// TwinCAT 3 PLC project MR1K4_PLC
// ProgramVersion: 3.1.4022.7
// libraries:
//   Tc2_SerialCom, * (Beckhoff Automation GmbH)
//   Tc2_Standard, * (Beckhoff Automation GmbH)
//   Tc2_System, * (Beckhoff Automation GmbH)
//   Tc2_Utilities, * (Beckhoff Automation GmbH)
//   Tc3_Module, * (Beckhoff Automation GmbH)
//   lcls-twincat-motion,1.1.0,SLAC
//   lcls-twincat-optics,0.0.0,SLAC
// project tree:
//   GVLs/ GVL_COM_Buffers.TcGVL (not stored), GVL_M1K4.TcGVL, GVL_M1K4_Constants.TcGVL (not stored), GVL_SerialIO.TcGVL
//   / PiezoDriver.TcTTO, PlcTask.TcTTO, SerialIO.TcTTO
//   POUs/ Main.TcPOU
//   POUs/Serial Comm/ PiezoSerial.TcPOU, P_Serial_Com.TcPOU
// real-time tasks:
//   TASK PlcTask: cycle T#10ms, priority 20, ADS port 350
//   TASK PiezoDriver: cycle T#1ms, priority 3, ADS port 351
//   TASK SerialIO: cycle T#2ms, priority 1, ADS port 352
// motion (NC):
//   TASK NC-Task 1 SAF: cycle T#2ms, priority 4, ADS port 501
//   TASK NC-Task 1 SVB: cycle T#10ms, priority 8, ADS port 511
//   AXIS M1K4-Yup (id 1)
//     General: UnitName=um
//     Dynamic: Acceleration=200, Deceleration=200, DelayTime=0.008
//     Velo: Maximum=200
//     OtherSettings: AllowMotionCmdToSlave=true
//     encoder EncType=29
//       EncPara: ScaleFactorNumerator=0.001, MaxCount=#xffffffff
//         SoftEndMinControl: Enable=true, Range=2700
//         SoftEndMaxControl: Enable=true, Range=27000
//         Inc: RefSoftSyncMask=#x0000ffff
//     drive DrvType=24
//       DrvPara: Inverse=true
//         Analog: VeloReferenz=488.28125, ScaleFactorActTorque=0.1
//         TimeComp: TaskDelayCycles=1
//     controller CtrType=2
//       CtrPara: PriorControlFactor=1
//         PosDiffControl: Range=100
//         PID: PosKp=50, PosExtKp=10, DeadBandPosition=0.3
//         Observer: BandWidth=20
//   AXIS M1K4-Ydwn (id 2)
//     General: UnitName=um
//     Dynamic: Acceleration=200, Deceleration=200, DelayTime=0.008
//     Velo: Maximum=200
//     OtherSettings: AllowMotionCmdToSlave=true
//     encoder EncType=29
//       EncPara: ScaleFactorNumerator=0.001, MaxCount=#xffffffff
//         SoftEndMinControl: Enable=true, Range=2400
//         SoftEndMaxControl: Enable=true, Range=26700
//         Inc: RefSoftSyncMask=#x0000ffff
//     drive DrvType=24
//       DrvPara: Inverse=true
//         Analog: VeloReferenz=488.28125, ScaleFactorActTorque=0.1
//         TimeComp: TaskDelayCycles=1
//     controller CtrType=2
//       CtrPara: PriorControlFactor=1
//         PosDiffControl: Range=100
//         PID: PosKp=50, PosExtKp=10, DeadBandPosition=0.3
//         Observer: BandWidth=20
//   AXIS M1K4-Xup (id 3)
//     General: UnitName=um
//     Dynamic: Acceleration=2000, Deceleration=2000, DelayTime=0.008
//     Velo: Maximum=1000
//     OtherSettings: AllowMotionCmdToSlave=true
//     encoder EncType=29
//       EncPara: ScaleFactorNumerator=0.001, MaxCount=#xffffffff
//         SoftEndMinControl: Enable=true, Range=23400
//         SoftEndMaxControl: Enable=true, Range=25700
//         Inc: RefSoftSyncMask=#x0000ffff
//     drive DrvType=24
//       Analog: VeloReferenz=1220.703125, ScaleFactorActTorque=0.1
//       TimeComp: TaskDelayCycles=1
//     controller CtrType=2
//       CtrPara: PriorControlFactor=1
//         PosDiffControl: Range=100
//         PID: PosKp=50, PosExtKp=50, DeadBandPosition=0.4
//         Observer: BandWidth=20
//   AXIS M1K4-Xdwn (id 4)
//     General: UnitName=um
//     Dynamic: Acceleration=2000, Deceleration=2000, DelayTime=0.008
//     Velo: Maximum=1000
//     OtherSettings: AllowMotionCmdToSlave=true
//     encoder EncType=29
//       EncPara: ScaleFactorNumerator=0.001, MaxCount=#xffffffff
//         SoftEndMinControl: Enable=true, Range=23400
//         SoftEndMaxControl: Enable=true, Range=25800
//         Inc: RefSoftSyncMask=#x0000ffff
//     drive DrvType=24
//       DrvPara: Inverse=true
//         Analog: VeloReferenz=1220.703125, ScaleFactorActTorque=0.1
//         TimeComp: TaskDelayCycles=1
//     controller CtrType=2
//       CtrPara: PriorControlFactor=1
//         PosDiffControl: Range=100
//         PID: PosKp=50, PosExtKp=50, DeadBandPosition=0.4
//         Observer: BandWidth=20
//   AXIS M1K4-Pitch (id 5)
//     General: UnitName=urad
//     Dynamic: Acceleration=390, Deceleration=390, DelayTime=0.008
//     Velo: Maximum=150
//     OtherSettings: AllowMotionCmdToSlave=true
//     encoder EncType=29
//       EncPara: ScaleFactorNumerator=0.001949317739, MaxCount=#xffffffff
//         SoftEndMinControl: Enable=true, Range=17200
//         SoftEndMaxControl: Enable=true, Range=21800
//         Inc: RefSoftSyncMask=#x0000ffff
//     drive DrvType=24
//       Analog: VeloReferenz=761.4522417, ScaleFactorActTorque=0.1
//       TimeComp: TaskDelayCycles=1
//     controller CtrType=2
//       CtrPara: PriorControlFactor=1
//         PosDiffControl: Range=150
//         PID: PosExtKp=1, DeadBandPosition=0.25
//         Observer: BandWidth=20
//   AXIS M1K4-Bender (id 6)
//     General: UnitName=um
//     Dynamic: Acceleration=100, Deceleration=100, DelayTime=0.008
//     Velo: Maximum=190
//     OtherSettings: AllowMotionCmdToSlave=true
//     encoder EncType=29
//       EncPara: ScaleFactorNumerator=0.001, MaxCount=#xffffffff
//         Inc: RefSoftSyncMask=#x0000ffff
//     drive DrvType=24
//       Analog: VeloReferenz=195.3125, ScaleFactorActTorque=0.1
//       TimeComp: TaskDelayCycles=1
//     controller CtrType=2
//       CtrPara: PriorControlFactor=1
//         PID: PosKp=10, PosExtKp=1, DeadBandPosition=0.04
//         Observer: BandWidth=20
// I/O:
//   DEVICE Device 1 (EtherCAT), AmsNetId 172.21.92.63.2.1
//     Term 1 (EK1200)
// variable links:
//   (this object) <-> Device 1 (EtherCAT)/Term 1 (EK1200)/Term 5 (EK1122)/Term 6 (EK1100)/EL5042_M1K4_Yupdwn
//     Enc/Inputs/In/nComState @bit 1 <-> WcState/InputToggle
//     Enc/Inputs/In/nComState <-> WcState/WcState
//     Enc/Inputs/In/nDataIn1 <-> FB Inputs Channel 1/Position
//     Enc/Inputs/In/nDataIn1 <-> FB Inputs Channel 2/Position
//     Enc/Inputs/In/nState1 @bit 12 <-> FB Inputs Channel 1/Status/Diag
//     Enc/Inputs/In/nState1 @bit 12 <-> FB Inputs Channel 2/Status/Diag
//     Enc/Inputs/In/nState1 @bit 1 <-> FB Inputs Channel 1/Status/Error
//     Enc/Inputs/In/nState1 @bit 1 <-> FB Inputs Channel 2/Status/Error
//     Enc/Inputs/In/nState1 @bit 14 <-> FB Inputs Channel 1/Status/Input cycle counter
//     Enc/Inputs/In/nState1 @bit 14 <-> FB Inputs Channel 2/Status/Input cycle counter
//     Enc/Inputs/In/nState1 @bit 2 <-> FB Inputs Channel 1/Status/Ready
//     Enc/Inputs/In/nState1 @bit 2 <-> FB Inputs Channel 2/Status/Ready
//     Enc/Inputs/In/nState1 @bit 13 <-> FB Inputs Channel 1/Status/TxPDO State
//     Enc/Inputs/In/nState1 @bit 13 <-> FB Inputs Channel 2/Status/TxPDO State
//     Enc/Inputs/In/nState1 <-> FB Inputs Channel 1/Status/Warning
//     Enc/Inputs/In/nState1 <-> FB Inputs Channel 2/Status/Warning
//   (this object) <-> Device 1 (EtherCAT)/Term 1 (EK1200)/Term 5 (EK1122)/Term 6 (EK1100)/EL7041-1000_M1K4_Yup
//     Drive/Inputs/In/nState1 @bit 3 <-> STM Status/Status/Error
//     Drive/Inputs/In/nState1 @bit 5 <-> STM Status/Status/Moving negative
//     Drive/Inputs/In/nState1 @bit 4 <-> STM Status/Status/Moving positive
//     Drive/Inputs/In/nState1 @bit 1 <-> STM Status/Status/Ready
//     Drive/Inputs/In/nState1 <-> STM Status/Status/Ready to enable
//     Drive/Inputs/In/nState1 @bit 6 <-> STM Status/Status/Torque reduced
//     Drive/Inputs/In/nState1 @bit 2 <-> STM Status/Status/Warning
//     Drive/Inputs/In/nState2 @bit 3 <-> STM Status/Status/Digital input 1
//     Drive/Inputs/In/nState2 @bit 4 <-> STM Status/Status/Digital input 2
//     Drive/Inputs/In/nState2 @bit 5 <-> STM Status/Status/Sync error
//     Drive/Inputs/In/nState2 @bit 7 <-> STM Status/Status/TxPDO Toggle
//     Drive/Inputs/In/nState4 @bit 1 <-> WcState/InputToggle
//     Drive/Inputs/In/nState4 <-> WcState/WcState
//     Drive/Outputs/Out/nCtrl1 <-> STM Control/Control/Enable
//     Drive/Outputs/Out/nCtrl1 @bit 2 <-> STM Control/Control/Reduce torque
//     Drive/Outputs/Out/nCtrl1 @bit 1 <-> STM Control/Control/Reset
//     Drive/Outputs/Out/nDataOut2[0] <-> STM Velocity/Velocity
//   (this object) <-> Device 1 (EtherCAT)/Term 1 (EK1200)/Term 5 (EK1122)/Term 6 (EK1100)/EL7041-1000_M1K4_Ydwn
//     Drive/Inputs/In/nState1 @bit 3 <-> STM Status/Status/Error
//     Drive/Inputs/In/nState1 @bit 5 <-> STM Status/Status/Moving negative
//     Drive/Inputs/In/nState1 @bit 4 <-> STM Status/Status/Moving positive
//     Drive/Inputs/In/nState1 @bit 1 <-> STM Status/Status/Ready
//     Drive/Inputs/In/nState1 <-> STM Status/Status/Ready to enable
//     Drive/Inputs/In/nState1 @bit 6 <-> STM Status/Status/Torque reduced
//     Drive/Inputs/In/nState1 @bit 2 <-> STM Status/Status/Warning
//     Drive/Inputs/In/nState2 @bit 3 <-> STM Status/Status/Digital input 1
//     Drive/Inputs/In/nState2 @bit 4 <-> STM Status/Status/Digital input 2
//     Drive/Inputs/In/nState2 @bit 5 <-> STM Status/Status/Sync error
//     Drive/Inputs/In/nState2 @bit 7 <-> STM Status/Status/TxPDO Toggle
//     Drive/Inputs/In/nState4 @bit 1 <-> WcState/InputToggle
//     Drive/Inputs/In/nState4 <-> WcState/WcState
//     Drive/Outputs/Out/nCtrl1 <-> STM Control/Control/Enable
//     Drive/Outputs/Out/nCtrl1 @bit 2 <-> STM Control/Control/Reduce torque
//     Drive/Outputs/Out/nCtrl1 @bit 1 <-> STM Control/Control/Reset
//     Drive/Outputs/Out/nDataOut2[0] <-> STM Velocity/Velocity
//   (this object) <-> Device 1 (EtherCAT)/Term 1 (EK1200)/Term 5 (EK1122)/Term 6 (EK1100)/EL5042_M1K4_Xupdwn
//     Enc/Inputs/In/nComState @bit 1 <-> WcState/InputToggle
//     Enc/Inputs/In/nComState <-> WcState/WcState
//     Enc/Inputs/In/nDataIn1 <-> FB Inputs Channel 1/Position
//     Enc/Inputs/In/nDataIn1 <-> FB Inputs Channel 2/Position
//     Enc/Inputs/In/nState1 @bit 12 <-> FB Inputs Channel 1/Status/Diag
//     Enc/Inputs/In/nState1 @bit 12 <-> FB Inputs Channel 2/Status/Diag
//     Enc/Inputs/In/nState1 @bit 1 <-> FB Inputs Channel 1/Status/Error
//     Enc/Inputs/In/nState1 @bit 1 <-> FB Inputs Channel 2/Status/Error
//     Enc/Inputs/In/nState1 @bit 14 <-> FB Inputs Channel 1/Status/Input cycle counter
//     Enc/Inputs/In/nState1 @bit 14 <-> FB Inputs Channel 2/Status/Input cycle counter
//     Enc/Inputs/In/nState1 @bit 2 <-> FB Inputs Channel 1/Status/Ready
//     Enc/Inputs/In/nState1 @bit 2 <-> FB Inputs Channel 2/Status/Ready
//     Enc/Inputs/In/nState1 @bit 13 <-> FB Inputs Channel 1/Status/TxPDO State
//     Enc/Inputs/In/nState1 @bit 13 <-> FB Inputs Channel 2/Status/TxPDO State
//     Enc/Inputs/In/nState1 <-> FB Inputs Channel 1/Status/Warning
//     Enc/Inputs/In/nState1 <-> FB Inputs Channel 2/Status/Warning
//   (this object) <-> Device 1 (EtherCAT)/Term 1 (EK1200)/Term 5 (EK1122)/Term 6 (EK1100)/EL7041-1000_M1K4_Xup
//     Drive/Inputs/In/nState1 @bit 3 <-> STM Status/Status/Error
//     Drive/Inputs/In/nState1 @bit 5 <-> STM Status/Status/Moving negative
//     Drive/Inputs/In/nState1 @bit 4 <-> STM Status/Status/Moving positive
//     Drive/Inputs/In/nState1 @bit 1 <-> STM Status/Status/Ready
//     Drive/Inputs/In/nState1 <-> STM Status/Status/Ready to enable
//     Drive/Inputs/In/nState1 @bit 6 <-> STM Status/Status/Torque reduced
//     Drive/Inputs/In/nState1 @bit 2 <-> STM Status/Status/Warning
//     Drive/Inputs/In/nState2 @bit 3 <-> STM Status/Status/Digital input 1
//     Drive/Inputs/In/nState2 @bit 4 <-> STM Status/Status/Digital input 2
//     Drive/Inputs/In/nState2 @bit 5 <-> STM Status/Status/Sync error
//     Drive/Inputs/In/nState2 @bit 7 <-> STM Status/Status/TxPDO Toggle
//     Drive/Inputs/In/nState4 @bit 1 <-> WcState/InputToggle
//     Drive/Inputs/In/nState4 <-> WcState/WcState
//     Drive/Outputs/Out/nCtrl1 <-> STM Control/Control/Enable
//     Drive/Outputs/Out/nCtrl1 @bit 2 <-> STM Control/Control/Reduce torque
//     Drive/Outputs/Out/nCtrl1 @bit 1 <-> STM Control/Control/Reset
//     Drive/Outputs/Out/nDataOut2[0] <-> STM Velocity/Velocity
//   (this object) <-> Device 1 (EtherCAT)/Term 1 (EK1200)/Term 5 (EK1122)/Term 6 (EK1100)/EL7041-1000_M1K4_Xdwn
//     Drive/Inputs/In/nState1 @bit 3 <-> STM Status/Status/Error
//     Drive/Inputs/In/nState1 @bit 5 <-> STM Status/Status/Moving negative
//     Drive/Inputs/In/nState1 @bit 4 <-> STM Status/Status/Moving positive
//     Drive/Inputs/In/nState1 @bit 1 <-> STM Status/Status/Ready
//     Drive/Inputs/In/nState1 <-> STM Status/Status/Ready to enable
//     Drive/Inputs/In/nState1 @bit 6 <-> STM Status/Status/Torque reduced
//     Drive/Inputs/In/nState1 @bit 2 <-> STM Status/Status/Warning
//     Drive/Inputs/In/nState2 @bit 3 <-> STM Status/Status/Digital input 1
//     Drive/Inputs/In/nState2 @bit 4 <-> STM Status/Status/Digital input 2
//     Drive/Inputs/In/nState2 @bit 5 <-> STM Status/Status/Sync error
//     Drive/Inputs/In/nState2 @bit 7 <-> STM Status/Status/TxPDO Toggle
//     Drive/Inputs/In/nState4 @bit 1 <-> WcState/InputToggle
//     Drive/Inputs/In/nState4 <-> WcState/WcState
//     Drive/Outputs/Out/nCtrl1 <-> STM Control/Control/Enable
//     Drive/Outputs/Out/nCtrl1 @bit 2 <-> STM Control/Control/Reduce torque
//     Drive/Outputs/Out/nCtrl1 @bit 1 <-> STM Control/Control/Reset
//     Drive/Outputs/Out/nDataOut2[0] <-> STM Velocity/Velocity
//   (this object) <-> Device 1 (EtherCAT)/Term 1 (EK1200)/Term 5 (EK1122)/Term 6 (EK1100)/EL5042_M1K4_PitchBender
//     Enc/Inputs/In/nComState @bit 1 <-> WcState/InputToggle
//     Enc/Inputs/In/nComState <-> WcState/WcState
//     Enc/Inputs/In/nDataIn1 <-> FB Inputs Channel 1/Position
//     Enc/Inputs/In/nDataIn1 <-> FB Inputs Channel 2/Position
//     Enc/Inputs/In/nState1 @bit 12 <-> FB Inputs Channel 1/Status/Diag
//     Enc/Inputs/In/nState1 @bit 12 <-> FB Inputs Channel 2/Status/Diag
//     Enc/Inputs/In/nState1 @bit 1 <-> FB Inputs Channel 1/Status/Error
//     Enc/Inputs/In/nState1 @bit 1 <-> FB Inputs Channel 2/Status/Error
//     Enc/Inputs/In/nState1 @bit 14 <-> FB Inputs Channel 1/Status/Input cycle counter
//     Enc/Inputs/In/nState1 @bit 14 <-> FB Inputs Channel 2/Status/Input cycle counter
//     Enc/Inputs/In/nState1 @bit 2 <-> FB Inputs Channel 1/Status/Ready
//     Enc/Inputs/In/nState1 @bit 2 <-> FB Inputs Channel 2/Status/Ready
//     Enc/Inputs/In/nState1 @bit 13 <-> FB Inputs Channel 1/Status/TxPDO State
//     Enc/Inputs/In/nState1 @bit 13 <-> FB Inputs Channel 2/Status/TxPDO State
//     Enc/Inputs/In/nState1 <-> FB Inputs Channel 1/Status/Warning
//     Enc/Inputs/In/nState1 <-> FB Inputs Channel 2/Status/Warning
//   (this object) <-> Device 1 (EtherCAT)/Term 1 (EK1200)/Term 5 (EK1122)/Term 6 (EK1100)/EL7041-1000_M1K4_PitchCoarse
//     Drive/Inputs/In/nState1 @bit 3 <-> STM Status/Status/Error
//     Drive/Inputs/In/nState1 @bit 5 <-> STM Status/Status/Moving negative
//     Drive/Inputs/In/nState1 @bit 4 <-> STM Status/Status/Moving positive
//     Drive/Inputs/In/nState1 @bit 1 <-> STM Status/Status/Ready
//     Drive/Inputs/In/nState1 <-> STM Status/Status/Ready to enable
//     Drive/Inputs/In/nState1 @bit 6 <-> STM Status/Status/Torque reduced
//     Drive/Inputs/In/nState1 @bit 2 <-> STM Status/Status/Warning
//     Drive/Inputs/In/nState2 @bit 3 <-> STM Status/Status/Digital input 1
//     Drive/Inputs/In/nState2 @bit 4 <-> STM Status/Status/Digital input 2
//     Drive/Inputs/In/nState2 @bit 5 <-> STM Status/Status/Sync error
//     Drive/Inputs/In/nState2 @bit 7 <-> STM Status/Status/TxPDO Toggle
//     Drive/Inputs/In/nState4 @bit 1 <-> WcState/InputToggle
//     Drive/Inputs/In/nState4 <-> WcState/WcState
//     Drive/Outputs/Out/nCtrl1 <-> STM Control/Control/Enable
//     Drive/Outputs/Out/nCtrl1 @bit 2 <-> STM Control/Control/Reduce torque
//     Drive/Outputs/Out/nCtrl1 @bit 1 <-> STM Control/Control/Reset
//     Drive/Outputs/Out/nDataOut2[0] <-> STM Velocity/Velocity
//   (this object) <-> Device 1 (EtherCAT)/Term 1 (EK1200)/Term 5 (EK1122)/Term 6 (EK1100)/EL7041-1000_M1K4_Bender
//     Drive/Inputs/In/nState1 @bit 3 <-> STM Status/Status/Error
//     Drive/Inputs/In/nState1 @bit 5 <-> STM Status/Status/Moving negative
//     Drive/Inputs/In/nState1 @bit 4 <-> STM Status/Status/Moving positive
//     Drive/Inputs/In/nState1 @bit 1 <-> STM Status/Status/Ready
//     Drive/Inputs/In/nState1 <-> STM Status/Status/Ready to enable
//     Drive/Inputs/In/nState1 @bit 6 <-> STM Status/Status/Torque reduced
//     Drive/Inputs/In/nState1 @bit 2 <-> STM Status/Status/Warning
//     Drive/Inputs/In/nState2 @bit 3 <-> STM Status/Status/Digital input 1
//     Drive/Inputs/In/nState2 @bit 4 <-> STM Status/Status/Digital input 2
//     Drive/Inputs/In/nState2 @bit 5 <-> STM Status/Status/Sync error
//     Drive/Inputs/In/nState2 @bit 7 <-> STM Status/Status/TxPDO Toggle
//     Drive/Inputs/In/nState4 @bit 1 <-> WcState/InputToggle
//     Drive/Inputs/In/nState4 <-> WcState/WcState
//     Drive/Outputs/Out/nCtrl1 <-> STM Control/Control/Enable
//     Drive/Outputs/Out/nCtrl1 @bit 2 <-> STM Control/Control/Reduce torque
//     Drive/Outputs/Out/nCtrl1 @bit 1 <-> STM Control/Control/Reset
//     Drive/Outputs/Out/nDataOut2[0] <-> STM Velocity/Velocity
//   MR1K4_PLC Instance <-> Device 1 (EtherCAT)/Term 1 (EK1200)/Term 5 (EK1122)/Term 6 (EK1100)/EL1004_M1K4_STO
//     PlcTask Inputs/Main.M1K4.fbRunHOMS.bSTOEnable1 <-> Channel 1/Input
//     PlcTask Inputs/Main.M1K4.fbRunHOMS.bSTOEnable2 <-> Channel 2/Input
//   MR1K4_PLC Instance <-> Device 1 (EtherCAT)/Term 1 (EK1200)/Term 5 (EK1122)/Term 6 (EK1100)/EL5042_M1K4_PitchBender
//     PlcTask Inputs/GVL_M1K4.M1K4_Pitch.diEncCnt <-> FB Inputs Channel 1/Position
//   MR1K4_PLC Instance <-> Device 1 (EtherCAT)/Term 1 (EK1200)/Term 5 (EK1122)/Term 6 (EK1100)/EL5042_M1K4_Xupdwn
//     PlcTask Inputs/Main.M1K4.fbRunHOMS.stXdwnEnc/Count <-> FB Inputs Channel 2/Position
//     PlcTask Inputs/Main.M1K4.fbRunHOMS.stXupEnc/Count <-> FB Inputs Channel 1/Position
//   MR1K4_PLC Instance <-> Device 1 (EtherCAT)/Term 1 (EK1200)/Term 5 (EK1122)/Term 6 (EK1100)/EL5042_M1K4_Yupdwn
//     PlcTask Inputs/Main.M1K4.fbRunHOMS.stYdwnEnc/Count <-> FB Inputs Channel 2/Position
//     PlcTask Inputs/Main.M1K4.fbRunHOMS.stYupEnc/Count <-> FB Inputs Channel 1/Position
//   MR1K4_PLC Instance <-> Device 1 (EtherCAT)/Term 1 (EK1200)/Term 5 (EK1122)/Term 6 (EK1100)/EL6001_M1K4_PitchFine
//     SerialIO Inputs/GVL_SerialIO.Serial_stComIn_M1K4/D[{0..21}] <-> COM Inputs/Data In {0..21}  (22 links)
//     SerialIO Inputs/GVL_SerialIO.Serial_stComIn_M1K4/Status <-> COM Inputs/Status
//     SerialIO Outputs/GVL_SerialIO.Serial_stComOut_M1K4/Ctrl <-> COM Outputs/Ctrl
//     SerialIO Outputs/GVL_SerialIO.Serial_stComOut_M1K4/D[{0..21}] <-> COM Outputs/Data Out {0..21}  (22 links)
//   MR1K4_PLC Instance <-> Device 1 (EtherCAT)/Term 1 (EK1200)/Term 5 (EK1122)/Term 6 (EK1100)/EL7041-1000_M1K4_Bender
//     PlcTask Inputs/Main.M6.bLimitBackwardEnable <-> STM Status/Status/Digital input 2
//     PlcTask Inputs/Main.M6.bLimitForwardEnable <-> STM Status/Status/Digital input 1
//   MR1K4_PLC Instance <-> Device 1 (EtherCAT)/Term 1 (EK1200)/Term 5 (EK1122)/Term 6 (EK1100)/EL7041-1000_M1K4_PitchCoarse
//     PlcTask Inputs/Main.M5.bLimitBackwardEnable <-> STM Status/Status/Digital input 2
//     PlcTask Inputs/Main.M5.bLimitForwardEnable <-> STM Status/Status/Digital input 1
//   MR1K4_PLC Instance <-> Device 1 (EtherCAT)/Term 1 (EK1200)/Term 5 (EK1122)/Term 6 (EK1100)/EL7041-1000_M1K4_Xdwn
//     PlcTask Inputs/Main.M4.bLimitBackwardEnable <-> STM Status/Status/Digital input 2
//     PlcTask Inputs/Main.M4.bLimitForwardEnable <-> STM Status/Status/Digital input 1
//   MR1K4_PLC Instance <-> Device 1 (EtherCAT)/Term 1 (EK1200)/Term 5 (EK1122)/Term 6 (EK1100)/EL7041-1000_M1K4_Xup
//     PlcTask Inputs/Main.M3.bLimitBackwardEnable <-> STM Status/Status/Digital input 2
//     PlcTask Inputs/Main.M3.bLimitForwardEnable <-> STM Status/Status/Digital input 1
//   MR1K4_PLC Instance <-> Device 1 (EtherCAT)/Term 1 (EK1200)/Term 5 (EK1122)/Term 6 (EK1100)/EL7041-1000_M1K4_Ydwn
//     PlcTask Inputs/Main.M2.bLimitBackwardEnable <-> STM Status/Status/Digital input 2
//     PlcTask Inputs/Main.M2.bLimitForwardEnable <-> STM Status/Status/Digital input 1
//   MR1K4_PLC Instance <-> Device 1 (EtherCAT)/Term 1 (EK1200)/Term 5 (EK1122)/Term 6 (EK1100)/EL7041-1000_M1K4_Yup
//     PlcTask Inputs/Main.M1.bLimitBackwardEnable <-> STM Status/Status/Digital input 2
//     PlcTask Inputs/Main.M1.bLimitForwardEnable <-> STM Status/Status/Digital input 1
//   MR1K4_PLC Instance <-> NC-Task 1 SAF/Axes/M1K4-Bender
//     PlcTask Inputs/Main.M6.Axis.NcToPlc <-> Outputs/ToPlc
//     PlcTask Outputs/Main.M6.Axis.PlcToNc <-> Inputs/FromPlc
//   MR1K4_PLC Instance <-> NC-Task 1 SAF/Axes/M1K4-Pitch
//     PlcTask Inputs/Main.M5.Axis.NcToPlc <-> Outputs/ToPlc
//     PlcTask Outputs/Main.M5.Axis.PlcToNc <-> Inputs/FromPlc
//   MR1K4_PLC Instance <-> NC-Task 1 SAF/Axes/M1K4-Xdwn
//     PlcTask Inputs/Main.M4.Axis.NcToPlc <-> Outputs/ToPlc
//     PlcTask Outputs/Main.M4.Axis.PlcToNc <-> Inputs/FromPlc
//   MR1K4_PLC Instance <-> NC-Task 1 SAF/Axes/M1K4-Xup
//     PlcTask Inputs/Main.M3.Axis.NcToPlc <-> Outputs/ToPlc
//     PlcTask Outputs/Main.M3.Axis.PlcToNc <-> Inputs/FromPlc
//   MR1K4_PLC Instance <-> NC-Task 1 SAF/Axes/M1K4-Ydwn
//     PlcTask Inputs/Main.M2.Axis.NcToPlc <-> Outputs/ToPlc
//     PlcTask Outputs/Main.M2.Axis.PlcToNc <-> Inputs/FromPlc
//   MR1K4_PLC Instance <-> NC-Task 1 SAF/Axes/M1K4-Yup
//     PlcTask Inputs/Main.M1.Axis.NcToPlc <-> Outputs/ToPlc
//     PlcTask Outputs/Main.M1.Axis.PlcToNc <-> Inputs/FromPlc

CONFIGURATION MR1K4_PLC
    RESOURCE PLC ON TwinCAT3
        TASK PiezoDriver(INTERVAL := T#1ms, PRIORITY := 3);
        TASK PlcTask(INTERVAL := T#10ms, PRIORITY := 20);
        TASK SerialIO(INTERVAL := T#2ms, PRIORITY := 1);
        PROGRAM PiezoSerial WITH PiezoDriver : PiezoSerial;
        PROGRAM MAIN WITH PlcTask : MAIN;
        PROGRAM P_Serial_Com WITH SerialIO : P_Serial_Com;
    END_RESOURCE
END_CONFIGURATION

// ---- GVLs/GVL_M1K4.TcGVL
{attribute 'qualified_only'}
VAR_GLOBAL
	// Pitch Mechanism:
	{attribute 'TcLinkTo' := '.diEncCnt:=TIIB[EL5042_M1K4_PitchBender]^FB Inputs Channel 1^Position'}
	M1K4_Pitch : HOMS_PitchMechanism := (ReqPosLimHi := 21700,
		                                 ReqPosLimLo := 17400,
		                                 diEncPosLimHi := 11132100,
		                                 diEncPosLimLo := 8926200);
END_VAR

// ---- GVLs/GVL_SerialIO.TcGVL
VAR_GLOBAL
	//Better have your inputs and outputs!
	// M1K4
	Serial_stComIn_M1K4   AT %I*	:	EL6inData22B (*KL6inData22B*);
	Serial_stComOut_M1K4  AT %Q*	:	EL6outData22B (*KL6outData22B*);
END_VAR

// ---- POUs/Serial Comm/PiezoSerial.TcPOU
PROGRAM PiezoSerial
VAR
	//PI Serial
	fbE621SerialDriver_M1K4 : FB_PI_E621_SerialDriver;
	rtInitParams_M1K4	:	R_TRIG;
	tonTimeoutRst_M1K4	: TON := (PT:=T#2S); //For timeout reset
END_VAR

//Piezo E-621
///////////////////////
fbE621SerialDriver_M1K4.i_xExecute := TRUE;
fbE621SerialDriver_M1K4.i_xExecute R= fbE621SerialDriver_M1K4.q_xDone;
fbE621SerialDriver_M1K4(iq_stPiezoAxis:= GVL_M1K4.M1K4_Pitch.Piezo,
		                iq_stSerialRXBuffer:= Serial_RXBuffer_M1K4,
		                iq_stSerialTXBuffer:= Serial_TXBuffer_M1K4);

END_PROGRAM

// ---- POUs/Main.TcPOU
PROGRAM Main
VAR
	// M1K4
	// Motors
	{attribute 'TcLinkTo' := '.bLimitForwardEnable:=TIIB[EL7041-1000_M1K4_Yup]^STM Status^Status^Digital input 1;
                              .bLimitBackwardEnable:=TIIB[EL7041-1000_M1K4_Yup]^STM Status^Status^Digital input 2'}
	{attribute 'pytmc' := '
		pv: MR1K4:KFE:MMS:YUP
	'}
	M1 : DUT_MotionStage := (fVelocity:=200, nEnableMode:=ENUM_StageEnableMode.ALWAYS); // M1K4 Yup
	fbMotionStage_m1 : FB_MotionStage;

	{attribute 'TcLinkTo' := '.bLimitForwardEnable:=TIIB[EL7041-1000_M1K4_Ydwn]^STM Status^Status^Digital input 1;
                              .bLimitBackwardEnable:=TIIB[EL7041-1000_M1K4_Ydwn]^STM Status^Status^Digital input 2'}
	{attribute 'pytmc' := '
		pv: MR1K4:KFE:MMS:YDWN
	'}
	M2 : DUT_MotionStage := (fVelocity:=200, nEnableMode:=ENUM_StageEnableMode.ALWAYS); // M1K4 Ydwn
	fbMotionStage_m2 : FB_MotionStage;

	{attribute 'TcLinkTo' := '.bLimitForwardEnable:=TIIB[EL7041-1000_M1K4_Xup]^STM Status^Status^Digital input 1;
                              .bLimitBackwardEnable:=TIIB[EL7041-1000_M1K4_Xup]^STM Status^Status^Digital input 2'}
	{attribute 'pytmc' := '
		pv: MR1K4:KFE:MMS:XUP
	'}
	M3 : DUT_MotionStage := (fVelocity:=1000, nEnableMode:=ENUM_StageEnableMode.ALWAYS); // M1K4 Xup
	fbMotionStage_m3 : FB_MotionStage;

	{attribute 'TcLinkTo' := '.bLimitForwardEnable:=TIIB[EL7041-1000_M1K4_Xdwn]^STM Status^Status^Digital input 1;
                              .bLimitBackwardEnable:=TIIB[EL7041-1000_M1K4_Xdwn]^STM Status^Status^Digital input 2'}
	{attribute 'pytmc' := '
		pv: MR1K4:KFE:MMS:XDWN
	'}
	M4 : DUT_MotionStage := (fVelocity:=1000, nEnableMode:=ENUM_StageEnableMode.ALWAYS); // M1K4 Xdwn
	fbMotionStage_m4 : FB_MotionStage;

	{attribute 'TcLinkTo' := '.bLimitForwardEnable:=TIIB[EL7041-1000_M1K4_PitchCoarse]^STM Status^Status^Digital input 1;
                              .bLimitBackwardEnable:=TIIB[EL7041-1000_M1K4_PitchCoarse]^STM Status^Status^Digital input 2'}
	{attribute 'pytmc' := '
		pv: MR1K4:KFE:MMS:PITCH
	'}
	M5 : DUT_MotionStage := (fVelocity := 150); // M1K4 Pitch Stepper

	{attribute 'TcLinkTo' := '.bLimitForwardEnable:=TIIB[EL7041-1000_M1K4_Bender]^STM Status^Status^Digital input 1;
                              .bLimitBackwardEnable:=TIIB[EL7041-1000_M1K4_Bender]^STM Status^Status^Digital input 2'}
	{attribute 'pytmc' := '
		pv: MR1K4:KFE:MMS:BENDER
	'}
	M6 : DUT_MotionStage; // M1K4 Bender
	fbMotionStage_m6 : FB_MotionStage;

	{attribute 'TcLinkTo' := '.fbRunHOMS.bSTOEnable1:=TIIB[EL1004_M1K4_STO]^Channel 1^Input;
                              .fbRunHOMS.bSTOEnable2:=TIIB[EL1004_M1K4_STO]^Channel 2^Input;
	                          .fbRunHOMS.stYupEnc.Count:=TIIB[EL5042_M1K4_Yupdwn]^FB Inputs Channel 1^Position;
	                          .fbRunHOMS.stYdwnEnc.Count:=TIIB[EL5042_M1K4_Yupdwn]^FB Inputs Channel 2^Position;
	                          .fbRunHOMS.stXupEnc.Count:=TIIB[EL5042_M1K4_Xupdwn]^FB Inputs Channel 1^Position;
	                          .fbRunHOMS.stXdwnEnc.Count:=TIIB[EL5042_M1K4_Xupdwn]^FB Inputs Channel 2^Position'}
	{attribute 'pytmc' := '
		pv: MR1K4:KFE
	'}
	M1K4 : DUT_HOMS;

	// Encoder Arrays/RMS Watch:
	{attribute 'pytmc' := '
		pv: MR1K4:KFE:Y_ENC
	'}
	fbYRMSErrorM1K4 : FB_RMSWatch;
	fMaxYRMSErrorM1K4 : LREAL;
	fMinYRMSErrorM1K4 : LREAL;

	{attribute 'pytmc' := '
		pv: MR1K4:KFE:X_ENC
	'}
	fbXRMSErrorM1K4 : FB_RMSWatch;
	fMaxXRMSErrorM1K4 : LREAL;
	fMinXRMSErrorM1K4 : LREAL;

	{attribute 'pytmc' := '
		pv: MR1K4:KFE:PITCH_ENC
	'}
	fbPitchRMSErrorM1K4 : FB_RMSWatch;
	fMaxPitchRMSErrorM1K4 : LREAL;
	fMinPitchRMSErrorM1K4 : LREAL;

	{attribute 'pytmc' := '
		pv: MR1K4:KFE:BENDER_ENC
	'}
	fbBenderRMSErrorM1K4 : FB_RMSWatch;
	fMaxBenderRMSErrorM1K4 : LREAL;
	fMinBenderRMSErrorM1K4 : LREAL;

	// Pitch Control
	fbM1K4PitchControl : FB_PitchControl;
	bM1K4PitchDone : BOOL;
	bM1K4PitchBusy : BOOL;
END_VAR

// M1L0
M1K4.fbRunHOMS(stYup:=M1,
               stYdwn:=M2,
               stXup:=M3,
               stXdwn:=M4,
               stPitch:=M5,
               stBender:=M6,
	           nYupEncRef:=GVL_M1K4_Constants.nYUP_ENC_REF,
               nYdwnEncRef:=GVL_M1K4_Constants.nYDWN_ENC_REF,
               nXupEncRef:=GVL_M1K4_Constants.nXUP_ENC_REF,
               nXdwnEncRef:=GVL_M1K4_Constants.nXDWN_ENC_REF,
			   bExecuteCoupleY:=M1K4.bExecuteCoupleY,
               bExecuteCoupleX:=M1K4.bExecuteCoupleX,
			   bExecuteDecoupleY:=M1K4.bExecuteDecoupleY,
               bExecuteDecoupleX:=M1K4.bExecuteDecoupleX,
               bGantryAlreadyCoupledY=>M1K4.bGantryAlreadyCoupledY,
               bGantryAlreadyCoupledX=>M1K4.bGantryAlreadyCoupledX,
               nCurrGantryY=>M1K4.nCurrGantryY,
               nCurrGantryX=>M1K4.nCurrGantryX);

// Convert nCurrGantry to um (smaller number) to read out in epics
M1K4.fCurrGantryY_um := LINT_TO_REAL(M1K4.nCurrGantryY) / 1000.0;
M1K4.fCurrGantryX_um := LINT_TO_REAL(M1K4.nCurrGantryX) / 1000.0;

// FB_MotionStage's for non-piezo axes
fbMotionStage_m1(stMotionStage:=M1);
fbMotionStage_m2(stMotionStage:=M2);
fbMotionStage_m3(stMotionStage:=M3);
fbMotionStage_m4(stMotionStage:=M4);
fbMotionStage_m6(stMotionStage:=M6);

// Calculate Pitch RMS Error:
fbYRMSErrorM1K4(stMotionStage:=M1,
	            fMaxRMSError=>fMaxYRMSErrorM1K4,
				fMinRMSError=>fMinYRMSErrorM1K4);

fbXRMSErrorM1K4(stMotionStage:=M3,
	            fMaxRMSError=>fMaxXRMSErrorM1K4,
				fMinRMSError=>fMinXRMSErrorM1K4);

fbPitchRMSErrorM1K4(stMotionStage:=M5,
	                fMaxRMSError=>fMaxPitchRMSErrorM1K4,
					fMinRMSError=>fMinPitchRMSErrorM1K4);

// Pitch Control
M5.fVelocity := 150.0;
fbM1K4PitchControl(Pitch:=GVL_M1K4.M1K4_Pitch,
				   Stepper:=M5,
				   lrCurrentSetpoint:=M5.fPosition,
                   q_bDone=>bM1K4PitchDone,
                   q_bBusy=>bM1K4PitchBusy);
// When STO hit, need to reset SP
IF NOT M5.bHardwareEnable THEN
	M5.fPosition := M5.stAxisStatus.fActPosition;
END_IF

END_PROGRAM

// ---- POUs/Serial Comm/P_Serial_Com.TcPOU
PROGRAM P_Serial_Com
VAR
	fbSerialLineControl_EL6001_M1K4: SerialLineControl;
END_VAR

//These are the global IOs...don't forget to copy your data into them

(* EL6001 Serial port 0 com function *)
fbSerialLineControl_EL6001_M1K4(Mode:= SERIALLINEMODE_EL6_22B (*SERIALLINEMODE_KL6_22B_STANDARD*),
						        pComIn:= ADR(Serial_stComIn_M1K4),
						   	    pComOut:=ADR(Serial_stComOut_M1K4),
						        SizeComIn:= SIZEOF(Serial_stComIn_M1K4),
						        TxBuffer:= Serial_TXBuffer_M1K4,
						        RxBuffer:= Serial_RXBuffer_M1K4,
						        Error=> ,
						        ErrorID=> );

END_PROGRAM
